FUNCTION_BLOCK EL2809
VAR
	{attribute addProperty Name "WcState"}
	_wcState : WcStateBase;
	{attribute addProperty Name "Info data"}
	_infoData : InfoDataBase;
	_io : EL2xx9_Data;
END_VAR

PROPERTY IO : REFERENCE TO EL2xx9_Data
GET
IO REF= _io;
END_GET
END_PROPERTY

PROPERTY WcState : REFERENCE TO WcStateBase
GET
WcState REF= _wcState;
END_GET
END_PROPERTY

END_FUNCTION_BLOCK

(* stored: Version 1.1.0.1, ProductVersion 3.1.4024.9
   POU EL2809: Id {a5d8806d-2fa9-0a34-239c-97db45246e10}, SpecialFunc None
   Property IO: Id {dabe339c-d34f-0432-1c50-ffea13e91256}
   Get Get: Id {64ae64bb-fe0a-0314-0b28-b1babe4a9feb}
   Property WcState: Id {79e72ae9-cdee-0c7c-0c98-f15809129862}
   Get Get: Id {a56bf126-d78b-00cb-1d5a-66711d2af6cb} *)
